FUNCTION_BLOCK FB_Processing
VAR_INPUT
	SensorInput	:	REAL;
END_VAR
VAR_OUTPUT
	
END_VAR
VAR_IN_OUT
	slot		:	INT;	
END_VAR
VAR
	
END_VAR

END_FUNCTION_BLOCK

(* stored: Version 1.1.0.1, ProductVersion 3.1.4024.12
   POU FB_Processing: Id {e6c1c698-a5ab-41a3-a94f-e6ef9684c89a}, SpecialFunc None *)
